TYPE WrappedComponentExample_Status EXTENDS TcoCore.TcoStruct :
STRUCT
    ProgressThrow : INT;
    ActionDescription : STRING;
END_STRUCT
END_TYPE

(* stored: Version 1.1.0.1, ProductVersion 3.1.4024.12
   DUT WrappedComponentExample_Status: Id {ea73d9a9-b277-0a53-03b9-1234f3b7bb6c} *)
